TYPE DigitalInput :
STRUCT
	in AT %I*	:	BIT;
END_STRUCT
END_TYPE

(* stored: Version 1.1.0.1, ProductVersion 3.1.4020.12
   DUT DigitalInput: Id {f6636f4c-810b-465e-9ad4-607ec4fabc8a} *)
